RoboDK station: 3D_Part_V4_Mesh.rdk

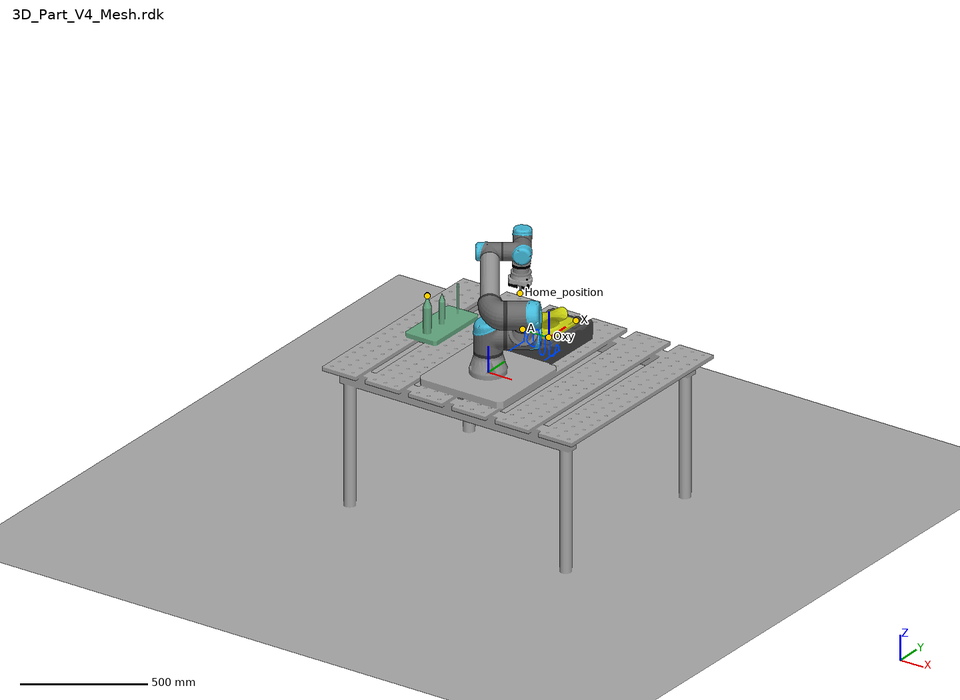
[picture v0: the station drawn from its stored meshes, robots at their saved joint values, targets as dots, program paths as lines]
Station 3D_Part_V4_Mesh (saved by RoboDK 5.6.0). Poses are relative to the parent item; angles as X-Y-Z fixed-axis rotations.
  - frame UR5e Base at (0, 0, 30) mm
    - target Home_position (joint target) at (21.87, 186.74, 274.06) mm, rotated rx 179.29 ry -1.86 rz -134.59 deg; joints [125.1, -36.39, -129.93, -103.31, 91.96, -190.29] of UR5e
    - robot UR5e: 6 axes, payload 5 kg, reach 850 mm, repeatability 0.03 mm, weight 18.4 kg
        modified DH rows (alpha deg, a mm, theta deg, d mm): 0, 0, 0, 162.5; 90, 0, 180, 0; 0, 425, 0, 0; 0, 392.25, 0, 133.3; -90, 0, 0, 99.7; 90, 0, 180, 99.6
        joint limits [-360, -360, -360, -360, -360, -360] to [360, 360, 360, 360, 360, 360]; home [0, -90, -90, 0, 90, 0]; saved at [125.1, -36.39, -129.93, -103.31, 91.96, -190.29]
      - tool Gripper, TCP at (0.02, 0, 134.54) mm, size 93 x 134.6 x 99.8 mm, geometry from UR5e
    - target 1_point_calibration_TCP (joint target) at (-409.67, 169.42, 149.93) mm, rotated rx 177.6 ry 0.93 rz 178.1 deg; joints [-38.601, -91.517, 122.976, -122.144, -92.477, -126.732] of UR5e
    - target 2_point_calibration_TCP (joint target) at (-410.25, 171.04, 150.5) mm, rotated rx 176.95 ry 38.31 rz 176.24 deg; joints [-30.106, -71.878, 98.621, -82.617, -108.81, -111.587] of UR5e
    - target 3_point_calibration_TCP (joint target) at (-409.99, 169.96, 150.21) mm, rotated rx 126.21 ry 38.31 rz 176.24 deg; joints [196.668, -105.719, -110.682, -107.023, 51.076, -69.389] of UR5e
    - target 4_point_calibration_TCP (joint target) at (-409.84, 170.1, 150.12) mm, rotated rx 173.91 ry -42.23 rz -175.16 deg; joints [-58.81, -99.027, 150.427, -169.407, -56.512, -142.715] of UR5e
    - target Oxy (Cartesian target) at (87.5, 290, 60) mm, rotated rx 180 ry 0 rz 180 deg; joints [99.313, -76.22, -149.564, -44.216, 90, -170.687] of UR5e
    - target X (Cartesian target) at (87.5, 475, 60) mm, rotated rx 180 ry 0 rz 180 deg; joints [95.58, -102.639, -123.551, -43.81, 90, -174.419] of UR5e
    - target A (Cartesian target) at (-37.5, 290, 60) mm, rotated rx 180 ry 0 rz 180 deg; joints [124.484, -73.976, -150.918, -45.106, 90, -145.515] of UR5e
  - object Table at (0, 200, 0) mm, size 1193.8 x 965.2 x 609.6 mm, geometry from Stol.stl
  - object Postolje_UR5e at (0, 0, 0) mm, rotated rx 90 ry 0 rz 0 deg, size 400 x 30 x 400 mm, geometry from Postolje_UR5e.STEP
  - object Sponge at (29.5, 380, 0) mm, rotated rx 90 ry 0 rz 0 deg, size 200 x 50.9 x 301 mm, geometry from sponge.STEP
  - object Sponge at (29.84, 379.94, 30) mm, rotated rx 90 ry 0 rz 0 deg, size 200 x 50.9 x 301 mm, geometry from sponge.STEP
  - object Calibration_Gauge at (-410, 270, 0) mm, rotated rx 0 ry 0 rz 90 deg, size 300 x 150 x 180 mm, geometry from kalibracijski_siljak_fiksni_3.stl
  - object Floor at (-40, 90, -610) mm, size 3000 x 3000 x 0 mm, geometry from Floor.stl
  - object 3D_Part at (25, 383, 190) mm, rotated rx 0 ry 0 rz -90 deg, size 200 x 145 x 75.1 mm, geometry from 3D_Part_V3.STEP
  - frame Frame_Part at (87.5, 290, 90) mm, rotated rx 0 ry 0 rz 90 deg
    - object Curves at (99, 61, -13.5) mm, rotated rx 0 ry 90 rz -90 deg
  - machining project Mesh settings: rotZ(0) | rotX(0)*rotY(0) | rotz(0) | onStart | onPathStart | onApproach | onPoint | onRetract | onFinish | SetRPM(%1) | SetTool(%1) | Extruder(%1) | default | default | OutOnMov(%1) | OutOffMov(%1) | onPathFinish | M_RunCode(%1)
  - program Mesh (153 instructions, listed below)
  - program Main_Program (5 instructions, listed below)
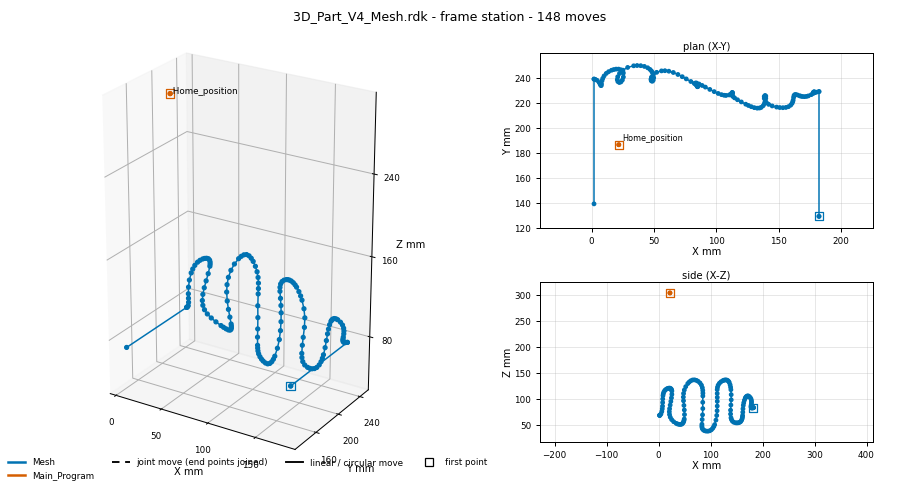
[picture p0: tool path of 3D_Part_V4_Mesh.rdk in frame station, 148 of 148 moves have a stored position in this frame; points joined in program order, loops and branches not executed]

--- program Mesh (robot UR5e) ---
  Smooth(1)
  Set speed (1000.0 mm/s)
  Set Ref.: Frame 2 -> Frame_Part
  Set Tool: Gripper
  Show Gripper
  MoveJ 1 to (-160.65, -94.79, -6.68) mm, rotated rx 0 ry 90 rz 0 deg; joints [113.018, -58.89, -133.638, -77.472, 90, -156.982]
  MoveL 2 to (-160.65, -94.79, -6.68) mm, rotated rx 0 ry 90 rz 0 deg; joints [113.018, -58.89, -133.638, -77.472, 90, -156.982]
  MoveL 3 to (-60.65, -94.79, -6.68) mm, rotated rx 0 ry 90 rz 0 deg; joints [113.018, -66.926, -145.826, -57.248, 90, -156.982]
  MoveL 4 to (-60.65, -94.79, -6.68) mm, rotated rx 0 ry 90 rz 0 deg; joints [113.018, -66.926, -145.826, -57.248, 90, -156.982]
  Set speed (50.0 mm/s)
  MoveL 5 to (-61.17, -92.68, -7.35) mm, rotated rx 0 ry 90 rz 0 deg; joints [112.972, -67.324, -145.539, -57.138, 90, -157.028]
  MoveL 6 to (-61.36, -91.56, -7.27) mm, rotated rx 0 ry 90 rz 0 deg; joints [112.863, -67.549, -145.391, -57.059, 90, -157.137]
  MoveL 7 to (-61.39, -90.76, -6.52) mm, rotated rx 0 ry 90 rz 0 deg; joints [112.647, -67.734, -145.293, -56.973, 90, -157.353]
  MoveL 8 to (-61.28, -90.5, -5.35) mm, rotated rx 0 ry 90 rz 0 deg; joints [112.394, -67.824, -145.265, -56.911, 90, -157.606]
  MoveL 9 to (-61.16, -90.49, -4.16) mm, rotated rx 0 ry 90 rz 0 deg; joints [112.158, -67.862, -145.267, -56.871, 90, -157.842]
  MoveL 10 to (-61, -90.65, -2.3) mm, rotated rx 0 ry 90 rz 0 deg; joints [111.802, -67.879, -145.287, -56.835, 90, -158.198]
  MoveL 11 to (-60.88, -91.02, 1.03) mm, rotated rx 0 ry 90 rz 0 deg; joints [111.169, -67.875, -145.308, -56.816, 90, -158.831]
  MoveL 12 to (-61.02, -91.2, 4) mm, rotated rx 0 ry 90 rz 0 deg; joints [110.59, -67.883, -145.281, -56.836, 90, -159.41]
  MoveL 13 to (-61.4, -91.04, 6.95) mm, rotated rx 0 ry 90 rz 0 deg; joints [109.987, -67.938, -145.185, -56.877, 90, -160.013]
  MoveL 14 to (-62.14, -90.23, 10.16) mm, rotated rx 0 ry 90 rz 0 deg; joints [109.286, -68.101, -144.972, -56.927, 90, -160.714]
  MoveL 15 to (-63.1, -88.63, 12.99) mm, rotated rx 0 ry 90 rz 0 deg; joints [108.609, -68.403, -144.647, -56.95, 90, -161.391]
  MoveL 16 to (-64.11, -86.29, 15.25) mm, rotated rx 0 ry 90 rz 0 deg; joints [108.005, -68.842, -144.239, -56.919, 90, -161.995]
  MoveL 17 to (-64.52, -84.79, 15.94) mm, rotated rx 0 ry 90 rz 0 deg; joints [107.775, -69.128, -144.014, -56.858, 90, -162.225]
  MoveL 18 to (-64.71, -83.11, 15.9) mm, rotated rx 0 ry 90 rz 0 deg; joints [107.676, -69.458, -143.802, -56.74, 90, -162.324]
  MoveL 19 to (-64.6, -81.47, 14.93) mm, rotated rx 0 ry 90 rz 0 deg; joints [107.763, -69.788, -143.641, -56.571, 90, -162.237]
  MoveL 20 to (-64.33, -80.23, 13.49) mm, rotated rx 0 ry 90 rz 0 deg; joints [107.966, -70.038, -143.55, -56.411, 90, -162.034]
  MoveL 21 to (-64.02, -79.27, 11.86) mm, rotated rx 0 ry 90 rz 0 deg; joints [108.219, -70.234, -143.494, -56.271, 90, -161.781]
  MoveL 22 to (-63.41, -77.6, 7.76) mm, rotated rx 0 ry 90 rz 0 deg; joints [108.899, -70.557, -143.421, -56.022, 90, -161.101]
  MoveL 23 to (-63.03, -76.3, 2.85) mm, rotated rx 0 ry 90 rz 0 deg; joints [109.747, -70.77, -143.367, -55.864, 90, -160.253]
  MoveL 24 to (-63.08, -75.43, -2.13) mm, rotated rx 0 ry 90 rz 0 deg; joints [110.628, -70.853, -143.31, -55.836, 90, -159.372]
  MoveL 25 to (-63.84, -74.78, -8.81) mm, rotated rx 0 ry 90 rz 0 deg; joints [111.832, -70.8, -143.207, -55.993, 90, -158.168]
  MoveL 26 to (-65.35, -74.45, -15.4) mm, rotated rx 0 ry 90 rz 0 deg; joints [113.032, -70.616, -143.046, -56.338, 90, -156.968]
  MoveL 27 to (-67.51, -74.1, -21.79) mm, rotated rx 0 ry 90 rz 0 deg; joints [114.18, -70.389, -142.797, -56.814, 90, -155.82]
  MoveL 28 to (-68.79, -73.76, -24.91) mm, rotated rx 0 ry 90 rz 0 deg; joints [114.722, -70.298, -142.626, -57.076, 90, -155.278]
  MoveL 29 to (-70.15, -73.17, -27.97) mm, rotated rx 0 ry 90 rz 0 deg; joints [115.226, -70.255, -142.413, -57.333, 90, -154.774]
  MoveL 30 to (-71.54, -72.12, -30.89) mm, rotated rx 0 ry 90 rz 0 deg; joints [115.664, -70.31, -142.141, -57.549, 90, -154.336]
  MoveL 31 to (-72.76, -70.3, -33.47) mm, rotated rx 0 ry 90 rz 0 deg; joints [115.968, -70.547, -141.795, -57.658, 90, -154.032]
  MoveL 32 to (-73.36, -68.28, -34.9) mm, rotated rx 0 ry 90 rz 0 deg; joints [116.046, -70.891, -141.492, -57.617, 90, -153.954]
  MoveL 33 to (-73.57, -65.88, -35.69) mm, rotated rx 0 ry 90 rz 0 deg; joints [115.98, -71.352, -141.187, -57.461, 90, -154.02]
  MoveL 34 to (-73.45, -63.35, -35.95) mm, rotated rx 0 ry 90 rz 0 deg; joints [115.811, -71.868, -140.901, -57.231, 90, -154.189]
  MoveL 35 to (-73.08, -60.84, -35.78) mm, rotated rx 0 ry 90 rz 0 deg; joints [115.572, -72.401, -140.643, -56.956, 90, -154.428]
  MoveL 36 to (-72.16, -57.29, -34.75) mm, rotated rx 0 ry 90 rz 0 deg; joints [115.106, -73.191, -140.317, -56.492, 90, -154.894]
  MoveL 37 to (-70.89, -54.44, -32.59) mm, rotated rx 0 ry 90 rz 0 deg; joints [114.515, -73.874, -140.11, -56.016, 90, -155.485]
  MoveL 38 to (-69.5, -52.68, -29.53) mm, rotated rx 0 ry 90 rz 0 deg; joints [113.861, -74.363, -140.041, -55.596, 90, -156.139]
  MoveL 39 to (-68.22, -51.73, -26.08) mm, rotated rx 0 ry 90 rz 0 deg; joints [113.205, -74.694, -140.054, -55.252, 90, -156.795]
  MoveL 40 to (-66.11, -50.95, -18.88) mm, rotated rx 0 ry 90 rz 0 deg; joints [111.923, -75.11, -140.158, -54.732, 90, -158.077]
  MoveL 41 to (-64.63, -50.92, -11.46) mm, rotated rx 0 ry 90 rz 0 deg; joints [110.647, -75.344, -140.269, -54.388, 90, -159.353]
  MoveL 42 to (-63.78, -51.56, -1.51) mm, rotated rx 0 ry 90 rz 0 deg; joints [108.961, -75.439, -140.358, -54.203, 90, -161.039]
  MoveL 43 to (-64.28, -52.17, 8.49) mm, rotated rx 0 ry 90 rz 0 deg; joints [107.246, -75.428, -140.274, -54.297, 90, -162.754]
  MoveL 44 to (-66.07, -52.16, 18.37) mm, rotated rx 0 ry 90 rz 0 deg; joints [105.504, -75.428, -139.953, -54.619, 90, -164.496]
  MoveL 45 to (-68.81, -51.57, 27.95) mm, rotated rx 0 ry 90 rz 0 deg; joints [103.785, -75.465, -139.439, -55.096, 90, -166.215]
  MoveL 46 to (-70.39, -51.01, 32.65) mm, rotated rx 0 ry 90 rz 0 deg; joints [102.929, -75.527, -139.118, -55.355, 90, -167.071]
  MoveL 47 to (-71.97, -50.08, 37.33) mm, rotated rx 0 ry 90 rz 0 deg; joints [102.068, -75.664, -138.745, -55.591, 90, -167.932]
  MoveL 48 to (-73.36, -48.44, 41.92) mm, rotated rx 0 ry 90 rz 0 deg; joints [101.202, -75.957, -138.3, -55.743, 90, -168.798]
  MoveL 49 to (-73.83, -47.12, 44.05) mm, rotated rx 0 ry 90 rz 0 deg; joints [100.785, -76.213, -138.042, -55.745, 90, -169.215]
  MoveL 50 to (-73.95, -45.28, 45.79) mm, rotated rx 0 ry 90 rz 0 deg; joints [100.422, -76.587, -137.762, -55.65, 90, -169.578]
  MoveL 51 to (-73.55, -42.96, 46.71) mm, rotated rx 0 ry 90 rz 0 deg; joints [100.19, -77.071, -137.495, -55.434, 90, -169.81]
  MoveL 52 to (-72.75, -40.55, 46.74) mm, rotated rx 0 ry 90 rz 0 deg; joints [100.111, -77.579, -137.275, -55.146, 90, -169.889]
  MoveL 53 to (-71.79, -38.26, 46.24) mm, rotated rx 0 ry 90 rz 0 deg; joints [100.127, -78.063, -137.097, -54.84, 90, -169.873]
  MoveL 54 to (-70.78, -36.1, 45.38) mm, rotated rx 0 ry 90 rz 0 deg; joints [100.207, -78.516, -136.948, -54.536, 90, -169.793]
  MoveL 55 to (-68.94, -32.56, 43.22) mm, rotated rx 0 ry 90 rz 0 deg; joints [100.46, -79.253, -136.73, -54.016, 90, -169.54]
  MoveL 56 to (-67.2, -29.47, 40.38) mm, rotated rx 0 ry 90 rz 0 deg; joints [100.835, -79.88, -136.571, -53.549, 90, -169.165]
  MoveL 57 to (-65.69, -27.12, 36.81) mm, rotated rx 0 ry 90 rz 0 deg; joints [101.348, -80.341, -136.492, -53.167, 90, -168.652]
  MoveL 58 to (-64.52, -25.75, 32.63) mm, rotated rx 0 ry 90 rz 0 deg; joints [101.986, -80.587, -136.515, -52.898, 90, -168.014]
  MoveL 59 to (-63.67, -25.25, 28.18) mm, rotated rx 0 ry 90 rz 0 deg; joints [102.695, -80.657, -136.617, -52.727, 90, -167.305]
  MoveL 60 to (-62.65, -25.26, 20.67) mm, rotated rx 0 ry 90 rz 0 deg; joints [103.918, -80.601, -136.848, -52.551, 90, -166.082]
  MoveL 61 to (-61.91, -25.37, 13.14) mm, rotated rx 0 ry 90 rz 0 deg; joints [105.147, -80.523, -137.045, -52.432, 90, -164.853]
  MoveL 62 to (-61.47, -25.39, 5.58) mm, rotated rx 0 ry 90 rz 0 deg; joints [106.373, -80.447, -137.184, -52.369, 90, -163.627]
  MoveL 63 to (-61.39, -25.29, -3.51) mm, rotated rx 0 ry 90 rz 0 deg; joints [107.835, -80.357, -137.268, -52.375, 90, -162.165]
  MoveL 64 to (-61.8, -25.02, -12.58) mm, rotated rx 0 ry 90 rz 0 deg; joints [109.273, -80.275, -137.256, -52.469, 90, -160.727]
  MoveL 65 to (-62.55, -24.31, -21.61) mm, rotated rx 0 ry 90 rz 0 deg; joints [110.665, -80.264, -137.126, -52.61, 90, -159.335]
  MoveL 66 to (-63.35, -22.82, -30.55) mm, rotated rx 0 ry 90 rz 0 deg; joints [111.977, -80.419, -136.859, -52.721, 90, -158.023]
  MoveL 67 to (-63.75, -20.31, -39.27) mm, rotated rx 0 ry 90 rz 0 deg; joints [113.163, -80.825, -136.471, -52.704, 90, -156.837]
  MoveL 68 to (-63.6, -18.73, -42.9) mm, rotated rx 0 ry 90 rz 0 deg; joints [113.612, -81.13, -136.258, -52.612, 90, -156.388]
  MoveL 69 to (-63.11, -16.66, -46.3) mm, rotated rx 0 ry 90 rz 0 deg; joints [113.987, -81.556, -136.009, -52.434, 90, -156.013]
  MoveL 70 to (-62.15, -14.01, -49.16) mm, rotated rx 0 ry 90 rz 0 deg; joints [114.238, -82.131, -135.724, -52.145, 90, -155.762]
  MoveL 71 to (-60.7, -10.82, -51.09) mm, rotated rx 0 ry 90 rz 0 deg; joints [114.311, -82.839, -135.412, -51.749, 90, -155.689]
  MoveL 72 to (-58.92, -7.3, -51.89) mm, rotated rx 0 ry 90 rz 0 deg; joints [114.196, -83.621, -135.09, -51.289, 90, -155.804]
  MoveL 73 to (-57.07, -3.74, -51.7) mm, rotated rx 0 ry 90 rz 0 deg; joints [113.937, -84.402, -134.77, -50.828, 90, -156.063]
  MoveL 74 to (-55.75, -1.13, -50.95) mm, rotated rx 0 ry 90 rz 0 deg; joints [113.663, -84.959, -134.534, -50.507, 90, -156.337]
  MoveL 75 to (-54.6, 1.31, -49.59) mm, rotated rx 0 ry 90 rz 0 deg; joints [113.315, -85.463, -134.308, -50.229, 90, -156.685]
  MoveL 76 to (-53.86, 3.23, -47.38) mm, rotated rx 0 ry 90 rz 0 deg; joints [112.883, -85.826, -134.124, -50.05, 90, -157.117]
  MoveL 77 to (-53.76, 4.07, -44.5) mm, rotated rx 0 ry 90 rz 0 deg; joints [112.42, -85.946, -134.036, -50.019, 90, -157.58]
  MoveL 78 to (-54.01, 4.22, -41.48) mm, rotated rx 0 ry 90 rz 0 deg; joints [111.979, -85.918, -134.013, -50.069, 90, -158.021]
  MoveL 79 to (-54.33, 4.16, -38.47) mm, rotated rx 0 ry 90 rz 0 deg; joints [111.55, -85.855, -134.009, -50.136, 90, -158.45]
  MoveL 80 to (-55.31, 3.66, -29.45) mm, rotated rx 0 ry 90 rz 0 deg; joints [110.271, -85.636, -134.02, -50.344, 90, -159.729]
  MoveL 81 to (-56.11, 2.97, -20.43) mm, rotated rx 0 ry 90 rz 0 deg; joints [108.988, -85.439, -134.043, -50.518, 90, -161.012]
  MoveL 82 to (-56.71, 2.49, -8.38) mm, rotated rx 0 ry 90 rz 0 deg; joints [107.231, -85.351, -134.008, -50.64, 90, -162.769]
  MoveL 83 to (-56.78, 2.59, 3.7) mm, rotated rx 0 ry 90 rz 0 deg; joints [105.426, -85.474, -133.886, -50.64, 90, -164.574]
  MoveL 84 to (-56.49, 2.4, 15.78) mm, rotated rx 0 ry 90 rz 0 deg; joints [103.623, -85.648, -133.784, -50.567, 90, -166.377]
  MoveL 85 to (-56.26, 2.3, 21.15) mm, rotated rx 0 ry 90 rz 0 deg; joints [102.818, -85.755, -133.733, -50.512, 90, -167.182]
  MoveL 86 to (-55.88, 2.52, 26.5) mm, rotated rx 0 ry 90 rz 0 deg; joints [102.005, -85.938, -133.64, -50.422, 90, -167.995]
  MoveL 87 to (-55.25, 3.35, 31.77) mm, rotated rx 0 ry 90 rz 0 deg; joints [101.187, -86.25, -133.478, -50.272, 90, -168.813]
  MoveL 88 to (-54.18, 5.09, 36.7) mm, rotated rx 0 ry 90 rz 0 deg; joints [100.396, -86.751, -133.223, -50.026, 90, -169.604]
  MoveL 89 to (-52.58, 7.9, 40.93) mm, rotated rx 0 ry 90 rz 0 deg; joints [99.691, -87.46, -132.872, -49.668, 90, -170.309]
  MoveL 90 to (-50.49, 11.6, 44.18) mm, rotated rx 0 ry 90 rz 0 deg; joints [99.119, -88.328, -132.45, -49.221, 90, -170.881]
  MoveL 91 to (-48.73, 14.78, 45.91) mm, rotated rx 0 ry 90 rz 0 deg; joints [98.791, -89.038, -132.104, -48.858, 90, -171.209]
  MoveL 92 to (-46.94, 18.25, 46.87) mm, rotated rx 0 ry 90 rz 0 deg; joints [98.576, -89.768, -131.733, -48.499, 90, -171.424]
  MoveL 93 to (-45.36, 21.94, 46.66) mm, rotated rx 0 ry 90 rz 0 deg; joints [98.526, -90.468, -131.34, -48.192, 90, -171.474]
  MoveL 94 to (-44.33, 25.52, 45.13) mm, rotated rx 0 ry 90 rz 0 deg; joints [98.667, -91.049, -130.951, -48, 90, -171.333]
  MoveL 95 to (-43.94, 28.68, 42.69) mm, rotated rx 0 ry 90 rz 0 deg; joints [98.943, -91.473, -130.589, -47.937, 90, -171.057]
  MoveL 96 to (-44.08, 31.4, 39.73) mm, rotated rx 0 ry 90 rz 0 deg; joints [99.297, -91.763, -130.26, -47.977, 90, -170.703]
  MoveL 97 to (-45.23, 35.31, 33.78) mm, rotated rx 0 ry 90 rz 0 deg; joints [100.032, -92.039, -129.744, -48.217, 90, -169.968]
  MoveL 98 to (-47.08, 38.01, 27.4) mm, rotated rx 0 ry 90 rz 0 deg; joints [100.844, -92.077, -129.345, -48.579, 90, -169.156]
  MoveL 99 to (-49.13, 39.48, 20.66) mm, rotated rx 0 ry 90 rz 0 deg; joints [101.729, -91.933, -129.097, -48.97, 90, -168.271]
  MoveL 100 to (-50.9, 39.88, 13.73) mm, rotated rx 0 ry 90 rz 0 deg; joints [102.664, -91.69, -129.008, -49.301, 90, -167.336]
  MoveL 101 to (-52.05, 39.58, 6.65) mm, rotated rx 0 ry 90 rz 0 deg; joints [103.639, -91.435, -129.053, -49.512, 90, -166.361]
  MoveL 102 to (-52.39, 38.77, -2.26) mm, rotated rx 0 ry 90 rz 0 deg; joints [104.88, -91.202, -129.228, -49.57, 90, -165.12]
  MoveL 103 to (-51.51, 38.03, -11.11) mm, rotated rx 0 ry 90 rz 0 deg; joints [106.109, -91.141, -129.461, -49.398, 90, -163.891]
  MoveL 104 to (-49.53, 37.69, -19.87) mm, rotated rx 0 ry 90 rz 0 deg; joints [107.309, -91.287, -129.691, -49.022, 90, -162.691]
  MoveL 105 to (-46.65, 38.13, -28.39) mm, rotated rx 0 ry 90 rz 0 deg; joints [108.434, -91.676, -129.848, -48.476, 90, -161.566]
  MoveL 106 to (-45.5, 38.62, -31.12) mm, rotated rx 0 ry 90 rz 0 deg; joints [108.778, -91.88, -129.859, -48.261, 90, -161.222]
  MoveL 107 to (-44.25, 39.4, -33.74) mm, rotated rx 0 ry 90 rz 0 deg; joints [109.092, -92.139, -129.832, -48.029, 90, -160.908]
  MoveL 108 to (-42.92, 40.62, -36.14) mm, rotated rx 0 ry 90 rz 0 deg; joints [109.353, -92.469, -129.745, -47.786, 90, -160.647]
  MoveL 109 to (-41.57, 42.51, -38.04) mm, rotated rx 0 ry 90 rz 0 deg; joints [109.516, -92.891, -129.559, -47.55, 90, -160.484]
  MoveL 110 to (-40.49, 45.14, -38.95) mm, rotated rx 0 ry 90 rz 0 deg; joints [109.513, -93.377, -129.248, -47.374, 90, -160.487]
  MoveL 111 to (-39.91, 48.09, -38.79) mm, rotated rx 0 ry 90 rz 0 deg; joints [109.357, -93.839, -128.858, -47.302, 90, -160.643]
  MoveL 112 to (-39.78, 50.97, -37.98) mm, rotated rx 0 ry 90 rz 0 deg; joints [109.122, -94.236, -128.447, -47.317, 90, -160.878]
  MoveL 113 to (-39.99, 53.7, -36.79) mm, rotated rx 0 ry 90 rz 0 deg; joints [108.848, -94.569, -128.034, -47.397, 90, -161.152]
  MoveL 114 to (-41.31, 58.54, -33.59) mm, rotated rx 0 ry 90 rz 0 deg; joints [108.231, -95.047, -127.237, -47.716, 90, -161.769]
  MoveL 115 to (-43.5, 62.38, -29.57) mm, rotated rx 0 ry 90 rz 0 deg; joints [107.563, -95.296, -126.524, -48.18, 90, -162.437]
  MoveL 116 to (-46.15, 65.07, -24.95) mm, rotated rx 0 ry 90 rz 0 deg; joints [106.873, -95.354, -125.941, -48.705, 90, -163.127]
  MoveL 117 to (-48.81, 66.51, -19.83) mm, rotated rx 0 ry 90 rz 0 deg; joints [106.172, -95.258, -125.534, -49.208, 90, -163.828]
  MoveL 118 to (-51.08, 66.84, -14.33) mm, rotated rx 0 ry 90 rz 0 deg; joints [105.465, -95.073, -125.306, -49.621, 90, -164.535]
  MoveL 119 to (-52.65, 66.37, -8.59) mm, rotated rx 0 ry 90 rz 0 deg; joints [104.753, -94.868, -125.237, -49.895, 90, -165.247]
  MoveL 120 to (-53.39, 65.24, -1.61) mm, rotated rx 0 ry 90 rz 0 deg; joints [103.9, -94.683, -125.302, -50.015, 90, -166.1]
  MoveL 121 to (-52.92, 63.93, 5.39) mm, rotated rx 0 ry 90 rz 0 deg; joints [103.042, -94.619, -125.463, -49.918, 90, -166.958]
  MoveL 122 to (-51.39, 62.78, 12.22) mm, rotated rx 0 ry 90 rz 0 deg; joints [102.195, -94.7, -125.665, -49.634, 90, -167.805]
  MoveL 123 to (-48.98, 61.98, 18.89) mm, rotated rx 0 ry 90 rz 0 deg; joints [101.353, -94.937, -125.863, -49.2, 90, -168.647]
  MoveL 124 to (-45.91, 62.02, 25.34) mm, rotated rx 0 ry 90 rz 0 deg; joints [100.515, -95.37, -125.97, -48.66, 90, -169.485]
  MoveL 125 to (-44.97, 62.35, 27.06) mm, rotated rx 0 ry 90 rz 0 deg; joints [100.283, -95.543, -125.956, -48.502, 90, -169.717]
  MoveL 126 to (-44.03, 62.98, 28.71) mm, rotated rx 0 ry 90 rz 0 deg; joints [100.056, -95.753, -125.9, -48.347, 90, -169.944]
  MoveL 127 to (-43.16, 64.08, 30.12) mm, rotated rx 0 ry 90 rz 0 deg; joints [99.848, -96.013, -125.77, -48.217, 90, -170.152]
  MoveL 128 to (-42.65, 65.82, 30.91) mm, rotated rx 0 ry 90 rz 0 deg; joints [99.707, -96.306, -125.532, -48.161, 90, -170.293]
  MoveL 129 to (-42.66, 67.81, 30.9) mm, rotated rx 0 ry 90 rz 0 deg; joints [99.665, -96.559, -125.237, -48.204, 90, -170.335]
  MoveL 130 to (-43.01, 69.71, 30.42) mm, rotated rx 0 ry 90 rz 0 deg; joints [99.685, -96.756, -124.938, -48.306, 90, -170.315]
  MoveL 131 to (-43.57, 71.47, 29.66) mm, rotated rx 0 ry 90 rz 0 deg; joints [99.743, -96.906, -124.652, -48.442, 90, -170.257]
  MoveL 132 to (-44.7, 73.79, 28.16) mm, rotated rx 0 ry 90 rz 0 deg; joints [99.882, -97.055, -124.256, -48.689, 90, -170.118]
  MoveL 133 to (-46.08, 75.67, 26.3) mm, rotated rx 0 ry 90 rz 0 deg; joints [100.075, -97.118, -123.914, -48.967, 90, -169.925]
  MoveL 134 to (-48.1, 77.43, 23.38) mm, rotated rx 0 ry 90 rz 0 deg; joints [100.403, -97.087, -123.561, -49.352, 90, -169.597]
  MoveL 135 to (-50.1, 78.49, 20.13) mm, rotated rx 0 ry 90 rz 0 deg; joints [100.784, -96.97, -123.314, -49.715, 90, -169.216]
  MoveL 136 to (-51.92, 79.08, 16.66) mm, rotated rx 0 ry 90 rz 0 deg; joints [101.202, -96.814, -123.149, -50.037, 90, -168.798]
  MoveL 137 to (-54.44, 79.55, 10.15) mm, rotated rx 0 ry 90 rz 0 deg; joints [102.001, -96.544, -122.985, -50.472, 90, -167.999]
  MoveL 138 to (-55.8, 79.72, 3.27) mm, rotated rx 0 ry 90 rz 0 deg; joints [102.851, -96.364, -122.937, -50.699, 90, -167.149]
  MoveL 139 to (-55.81, 79.97, -3.72) mm, rotated rx 0 ry 90 rz 0 deg; joints [103.709, -96.345, -122.957, -50.698, 90, -166.291]
  MoveL 140 to (-54.97, 80.44, -8.89) mm, rotated rx 0 ry 90 rz 0 deg; joints [104.333, -96.463, -122.979, -50.558, 90, -165.667]
  MoveL 141 to (-53.53, 81.33, -13.9) mm, rotated rx 0 ry 90 rz 0 deg; joints [104.921, -96.704, -122.972, -50.324, 90, -165.079]
  MoveL 142 to (-51.7, 82.97, -18.6) mm, rotated rx 0 ry 90 rz 0 deg; joints [105.441, -97.089, -122.868, -50.042, 90, -164.559]
  MoveL 143 to (-50.88, 84.43, -20.64) mm, rotated rx 0 ry 90 rz 0 deg; joints [105.64, -97.358, -122.709, -49.933, 90, -164.36]
  MoveL 144 to (-50.65, 85.5, -21.39) mm, rotated rx 0 ry 90 rz 0 deg; joints [105.695, -97.516, -122.566, -49.918, 90, -164.305]
  Set speed (1000.0 mm/s)
  MoveL 145 to (-50.65, 85.5, -21.39) mm, rotated rx 0 ry 90 rz 0 deg; joints [105.695, -97.516, -122.566, -49.918, 90, -164.305]
  MoveL 146 to (-150.65, 85.5, -21.39) mm, rotated rx 0 ry 90 rz 0 deg; joints [105.695, -89.448, -114.018, -66.534, 90, -164.305]

--- program Main_Program (robot UR5e) ---
  Set Ref.: UR5e Base
  Set Tool: Gripper
  MoveJ (Home_position)
  Call Mesh
  MoveJ (Home_position)
